Staubli VAL3: onF5Event.pgx

program onF5Event()
  local bool l_bCheck
  local string l_sMessage
begin
  // look if the bButton is enable
  if bButton[4]
    //
    if workingMode()==1
      resetMotion()
      call tcp:checkPoint(l_bCheck)
      if l_bCheck
        call language:message(l_sMessage,203)
        call tcp:goToPoint(nIndexTool)
        logMsg("[VALlaser] INTERFACE:Go to the reference Point")
        call use:timerDialog(l_sMessage,2)
      endIf
    endIf
  endIf
end
